// TIA Portal V16 export
// export: Created 2025-08-01T13:38:02.887217Z, ExportSetting WithDefaults, DisplayName Totally Integrated Automation Portal, DisplayVersion V16, DisplayName TIA Portal Version Control Interface, DisplayVersion V16, DisplayName TIA Portal Openness, DisplayVersion V16, DisplayName STEP 7 Professional, DisplayVersion V16, DisplayName STEP 7 Safety, DisplayVersion V16, DisplayName WinCC Advanced, DisplayVersion V16
DATA_BLOCK "FB_Encoder64Bit_DB"   // DB92
VERSION : 0.1
// stored: AutoNumber true, InstanceOfName FB_Encoder64Bit, InstanceOfType FB
"FB_Encoder64Bit"
   // VAR_INPUT
   //    EncoderRaw : DInt;
   //    PulsFactor : Real;
   //    MaxRawValue : DInt;
   //    FirstCycle { ExternalVisible := 'False'; ExternalWritable := 'False'} : Bool;
   // END_VAR
   // VAR_OUTPUT
   //    TotalPulses : DInt;
   //    Total_mm : Real;
   //    GlobalCounter : DInt;
   //    SegmentCounter : DInt;
   // END_VAR
BEGIN
END_DATA_BLOCK
